// TIA Portal project "Hata_Belirleme_Kesmesi_Uygulaması_V1" (V16)

(* hardware
DEVICE "S7-1200 station_1"  S7-1200 Station
   slot 0: "Rack_0"  S7-1200 Rack  Rack  V1.0
   slot 1: "PLC_1"  CPU 1214C DC/DC/DC  6ES7 214-1AG40-0XB0  V4.4
   slot 2: "DI 8x24VDC_1"  6ES7 221-1BF32-0XB0  V2.0
   slot 3: "AI 4x13BIT_1"  6ES7 231-4HD32-0XB0  V2.1
   slot 4: "AQ 2x14BIT_1"  SM 1232 AQ2  6ES7 232-4HB32-0XB0  V2.1
*)

// ===== PLC "PLC_1"  CPU 1214C DC/DC/DC =====

DATA_BLOCK "Sistem Hataları"   // DB1
{ S7_Optimized_Access := 'TRUE' }
VERSION : 0.1
   VAR
      "Hata_Sebebi (I/O State)" : Word;
      "Hatalı_Modül (LADDR)" : Hw_Any;
      "Hatalı_Kanal (Channel)" : UInt;
      "Çoklu_Hata (MultiError)" : Bool;
   END_VAR
BEGIN
END_DATA_BLOCK

ORGANIZATION_BLOCK "Main"   // OB1, LAD, ProgramCycle
TITLE = "Main Program Sweep (Cycle)"
{ S7_Optimized_Access := 'TRUE' }
VERSION : 0.1
   VAR_INPUT
      Initial_Call : Bool;   // Initial call of this OB
      Remanence : Bool;   // =True, if remanent data are available
   END_VAR
BEGIN
END_ORGANIZATION_BLOCK

ORGANIZATION_BLOCK "Diagnostic error interrupt"   // OB82, LAD, DiagnosticErrorInterrupt
{ S7_Optimized_Access := 'TRUE' }
VERSION : 0.1
   VAR_INPUT
      IO_State : Word;   // IO state of the HW object
      LADDR : Hw_Any;   // Hardware identifier
      Channel : UInt;   // Channel number
      MultiError : Bool;   // =true if more than one error is present
   END_VAR
BEGIN

REGION Network 1: Hata Arama Programı
   // - PLC’de bir giriş/çıkış modülünde veya donanım kanalında teşhis hatası oluştuğunda otomatik çalışır ve hatanın nereden geldiğini programda kaydetmeni sağlar.
   // 
   // 
   // Senin programında:
   // 
   // 
   // IO_State → Donanımın hata durum bilgisini verir.
   // 
   // LADDR → Hatanın hangi donanım/modül adresinden geldiğini gösterir.
   // 
   // Channel → Hatalı kanal numarasını verir.
   // 
   // MultiError → Aynı anda birden fazla hata olup olmadığını bildirir.
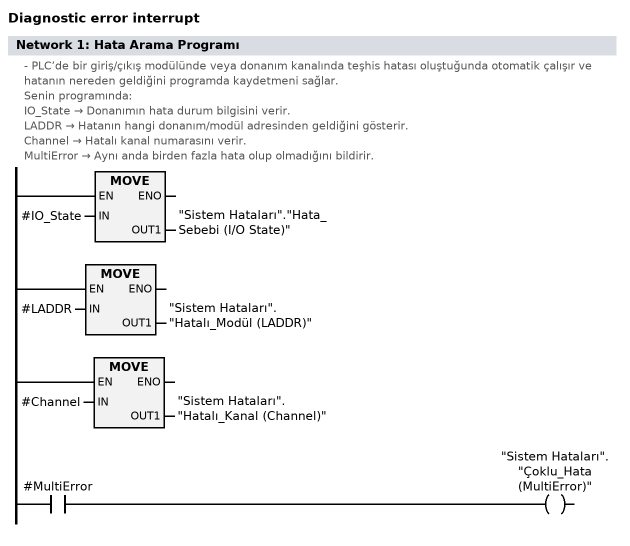
   RUNG wire#powerrail
      Move(in := #IO_State, out1 => "Sistem Hataları"."Hata_Sebebi (I/O State)")
   END_RUNG
   RUNG wire#powerrail
      Move(in := #LADDR, out1 => "Sistem Hataları"."Hatalı_Modül (LADDR)")
   END_RUNG
   RUNG wire#powerrail
      Move(in := #Channel, out1 => "Sistem Hataları"."Hatalı_Kanal (Channel)")
   END_RUNG
   RUNG wire#powerrail
      Contact( #MultiError )
      Coil( "Sistem Hataları"."Çoklu_Hata (MultiError)" )
   END_RUNG
   // the same network as SCL:
   "Sistem Hataları"."Hata_Sebebi (I/O State)" := #IO_State;
   "Sistem Hataları"."Hatalı_Modül (LADDR)" := #LADDR;
   "Sistem Hataları"."Hatalı_Kanal (Channel)" := #Channel;
   "Sistem Hataları"."Çoklu_Hata (MultiError)" := #MultiError;
END_REGION
END_ORGANIZATION_BLOCK